WHILE THIS^.fbStations.HasNextObject() DO
	IF __QUERYINTERFACE(THIS^.fbStations.GetNextObject(),ipEachStation) THEN
		//Return TRUE if found
		IF (ipEachStation.TargetGroupe = sStation) OR (ipEachStation.LUID = sStation) THEN
			CheckTargetExists := TRUE;
			EXIT;
		END_IF
	END_IF
END_WHILE

THIS^.fbStations.RestoreIterator();
END_METHOD

METHOD Station : I_XP_Station_PLC
VAR_INPUT
	sLUID : STRING;
END_VAR
//IF no station was found, INTERFACE is 0 -> can generate fatal error
__QUERYINTERFACE(THIS^.fbStations.FindLUID(sLUID),Station);
END_METHOD

METHOD LinkEnvironment : HRESULT
VAR_INPUT
	ipEnvironment : I_CH_Object;
END_VAR

VAR
	ipXpEnvironment : I_XP_Environment;
END_VAR
IF ipEnvironment <> 0 AND_THEN __QUERYINTERFACE(ipEnvironment,ipXpEnvironment) THEN
	THIS^.ipEnvironment := ipXpEnvironment;
ELSE
	LinkEnvironment := E_FAIL;
	THIS^.bErrorDuringFbInit := TRUE;
END_IF
END_METHOD

METHOD LinkGroup : HRESULT
VAR_INPUT
	ipGroup : I_CH_Object;
END_VAR

VAR
	ipXpGroup : I_XP_Group;
END_VAR
IF ipGroup <> 0 AND_THEN __QUERYINTERFACE(ipGroup,ipXpGroup) THEN
	THIS^.ipGroup := ipXpGroup;
ELSE
	LinkGroup := E_FAIL;
	THIS^.bErrorDuringFbInit := TRUE;
END_IF
END_METHOD

METHOD RegisterMover : HRESULT
VAR_INPUT
	ipMover : I_CH_Object;
END_VAR

VAR
	ipXpMover : I_XP_Mover;
END_VAR
IF ipMover = 0 THEN
	//Invalide interface	
	THIS^.bErrorDuringFbInit := TRUE;
	RegisterMover := E_FAIL;
	
ELSIF NOT __QUERYINTERFACE(ipMover, ipXpMover) THEN
	//The required interface is missing
	THIS^.bErrorDuringFbInit := TRUE;
	RegisterMover := E_FAIL;
	
ELSIF THIS^.fbMovers.IsFull THEN
	//List is full
	THIS^.bErrorDuringFbInit := TRUE;
	RegisterMover := E_FAIL;
	
ELSIF THIS^.bInitDone THEN
	//To late. System is initilized
	THIS^.bErrorDuringFbInit := TRUE;
	RegisterMover := E_FAIL;
	
ELSE
	
	THIS^.fbMovers.AddObject(ipMover);
END_IF
END_METHOD

METHOD RegisterStation : HRESULT
VAR_INPUT
	ipStation : I_CH_Object;
END_VAR

VAR
	ipXpStation : I_XP_Station;
END_VAR
IF ipStation = 0 THEN
	//Invalide interface	
	THIS^.bErrorDuringFbInit := TRUE;
	RegisterStation := E_FAIL;
	
ELSIF NOT __QUERYINTERFACE(ipStation, ipXpStation) THEN
	//The required interface is missing
	THIS^.bErrorDuringFbInit := TRUE;
	RegisterStation := E_FAIL;
	
ELSIF THIS^.fbStations.IsFull THEN
	//List is full
	THIS^.bErrorDuringFbInit := TRUE;
	RegisterStation := E_FAIL;
	
ELSIF THIS^.bInitDone THEN
	//To late. System is initilized
	THIS^.bErrorDuringFbInit := TRUE;
	RegisterStation := E_FAIL;
		
ELSE
	
	THIS^.fbStations.AddObject(ipStation);
END_IF
END_METHOD

METHOD RegisterTrack : HRESULT
VAR_INPUT
	ipTrack : I_CH_Object;
END_VAR

VAR
	ipXpTrack : I_XP_Track;
END_VAR
IF ipTrack = 0 THEN
	//Invalide interface	
	THIS^.bErrorDuringFbInit := TRUE;
	RegisterTrack := E_FAIL;
	
ELSIF NOT __QUERYINTERFACE(ipTrack, ipXpTrack) THEN
	//The required interface is missing
	THIS^.bErrorDuringFbInit := TRUE;
	RegisterTrack := E_FAIL;
	
ELSIF THIS^.fbTracks.IsFull THEN
	//List is full
	THIS^.bErrorDuringFbInit := TRUE;
	RegisterTrack := E_FAIL;
	
ELSIF THIS^.bInitDone THEN
	//To late. System is initilized
	THIS^.bErrorDuringFbInit := TRUE;
	RegisterTrack := E_FAIL;
		
ELSE
	
	THIS^.fbTracks.AddObject(ipTrack);
END_IF
END_METHOD

METHOD RegisterTrigger : HRESULT
VAR_INPUT
	ipTrigger	: CHALET_BaseComponents.I_CH_Object;
END_VAR
VAR
	ipXpTrigger : I_Xp_Trigger;
END_VAR
IF ipTrigger = 0 THEN
	//Invalide interface	
	THIS^.bErrorDuringFbInit := TRUE;
	RegisterTrigger := E_FAIL;
	
ELSIF NOT __QUERYINTERFACE(ipTrigger, ipXpTrigger) THEN
	//The required interface is missing
	THIS^.bErrorDuringFbInit := TRUE;
	RegisterTrigger := E_FAIL;
	
ELSIF THIS^.fbTriggers.IsFull THEN
	//List is full
	THIS^.bErrorDuringFbInit := TRUE;
	RegisterTrigger := E_FAIL;
	
ELSIF THIS^.bInitDone THEN
	//To late. System is initilized
	THIS^.bErrorDuringFbInit := TRUE;
	RegisterTrigger := E_FAIL;
		
ELSE
	
	THIS^.fbTriggers.AddObject(ipTrigger);
END_IF
END_METHOD

METHOD RegisterZone : HRESULT
VAR_INPUT
	ipZone	: CHALET_BaseComponents.I_CH_Object;
END_VAR
VAR
	ipXpsZone : I_XP_Zone;
END_VAR
IF ipZone = 0 THEN
	//Invalide interface	
	THIS^.bErrorDuringFbInit := TRUE;
	RegisterZone := E_FAIL;

ELSIF NOT __QUERYINTERFACE(ipZone, ipXpsZone) THEN
	//The required interface is missing
	THIS^.bErrorDuringFbInit := TRUE;
	RegisterZone := E_FAIL;
	
ELSIF THIS^.fbZones.IsFull THEN
	//List is full
	THIS^.bErrorDuringFbInit := TRUE;
	RegisterZone := E_FAIL;
	
ELSIF THIS^.bInitDone THEN
	//To late. System is initilized
	THIS^.bErrorDuringFbInit := TRUE;
	RegisterZone := E_FAIL;
		
ELSE
	
	THIS^.fbZones.AddObject(ipZone);	
END_IF
END_METHOD

{attribute 'monitoring':='call'}
PROPERTY Enviroment : I_XP_Environment
GET
Enviroment := THIS^.ipEnvironment;
END_GET
END_PROPERTY

METHOD FB_init : BOOL
VAR_INPUT
	bInitRetains : BOOL; // if TRUE, the retain variables are initialized (warm start / cold start)
	bInCopyCode : BOOL;  // if TRUE, the instance afterwards gets moved into the copy code (online change)
	
	METAdsPort : UINT; 
END_VAR
VAR
	fbGetCurTaskIdx  : GETCURTASKINDEX;
END_VAR
THIS^.nMETAdsPort := METAdsPort;
END_METHOD

{attribute 'monitoring':='call'}
PROPERTY Feedback : CHALET_BaseComponents.I_CH_Feedback
GET
Feedback := THIS^.fbFeedback;
END_GET
END_PROPERTY

{attribute 'monitoring':='call'}
PROPERTY METAdsPort : UINT
GET
METAdsPort := nMETAdsPort;
END_GET
END_PROPERTY

{attribute 'monitoring':='call'}
PROPERTY Movers : CHALET_BaseComponents.I_CH_LIST
GET
Movers := THIS^.fbMovers;
END_GET
END_PROPERTY

{attribute 'monitoring':='call'}
PROPERTY Stations : CHALET_BaseComponents.I_CH_LIST
GET
Stations := THIS^.fbStations;
END_GET
END_PROPERTY

{attribute 'monitoring':='call'}
PROPERTY Tracks : CHALET_BaseComponents.I_CH_LIST
GET
Tracks := THIS^.fbTracks;
END_GET
END_PROPERTY

{attribute 'monitoring':='call'}
PROPERTY Triggers : CHALET_BaseComponents.I_CH_LIST
GET
Triggers := THIS^.fbTriggers;
END_GET
END_PROPERTY

METHOD Update : HRESULT
VAR_INPUT
END_VAR
VAR
	hr : HRESULT;
END_VAR
//Force to do an init at beginn
IF NOT THIS^.Initialized THEN
	THIS^.Initialize();
	RETURN;
END_IF

hr := S_OK;

hr := GetMostSignificant(hr, THIS^.Enabling());
hr := GetMostSignificant(hr, THIS^.Disabling());




// ********************** Set feedback depending on active command *******************************
IF THIS^.eActiveCommand <> E_NcAxisCommands.None THEN
	fbFeedback.ActiveCommand 	:= TO_STRING(THIS^.eActiveCommand);	
END_IF

CASE THIS^.eActiveCommand OF
	E_NcAxisCommands.None: 
		;

	E_NcAxisCommands.Initialize:
		fbFeedback.Busy 		:= NOT THIS^.bInitDone;
		fbFeedback.Done 		:= THIS^.bInitDone;
		fbFeedback.ErrorId 		:= 0;
		
	E_NcAxisCommands.Enable:
		fbFeedback.Busy 		:= nSeqEnabling > 0;
		fbFeedback.Done 		:= THIS^.Enabled;
		IF nSeqEnabling > 1000 THEN
			fbFeedback.ErrorId 		:= nSeqEnabling;
		END_IF
		
	E_NcAxisCommands.Disable:
		fbFeedback.Busy 		:= nSeqDisabling > 0;
		fbFeedback.Done 		:= THIS^.Disabled;
		IF nSeqDisabling > 1000 THEN
			fbFeedback.ErrorId 		:= nSeqDisabling;
		END_IF
		


	ELSE//External command in subclass
		;
END_CASE


// **********************  Stop to execute commands on .done or .error ***************************
IF fbFeedback.Done OR THIS^.fbFeedback.Error THEN
	eActiveCommand 				:= E_NcAxisCommands.None;
END_IF







hr := GetMostSignificant(hr, THIS^.fbMovers.Update());
hr := GetMostSignificant(hr, THIS^.fbTracks.Update());
hr := GetMostSignificant(hr, THIS^.fbStations.Update());
hr := GetMostSignificant(hr, THIS^.fbZones.Update());
hr := GetMostSignificant(hr, THIS^.fbTriggers.Update());
hr := GetMostSignificant(hr, THIS^.ipGroup.Update());
hr := GetMostSignificant(hr, THIS^.ipEnvironment.Update());


Update:= hr;
END_METHOD

{attribute 'monitoring':='call'}
PROPERTY Zones : CHALET_BaseComponents.I_CH_LIST
GET
Zones := THIS^.fbZones;
END_GET
END_PROPERTY

END_FUNCTION_BLOCK

// COMPONENTs/Track/FB_XP_Track
{attribute 'no_explicit_call' := 'Do not call the body - Stick to OOP'}
(* XPlanar track - n per associated XPlanar. Can be instantiated as an array and/or individually
	The Planar track is a software object that represents a (virtual) one-dimensional path on the two-dimensional XPlanar stator surface. 
	Several Planar movers can be lined up and moved on this path. Collisions are prevented by keeping a preset distance between the movers. *)	
FUNCTION_BLOCK FB_XP_Track EXTENDS FB_CH_Object IMPLEMENTS I_XP_Track
VAR
	//Link to Planar-Track object
	fbTrack : MC_PlanarTrack;
	
	{attribute 'hide'}  
	bInitDone :BOOL := FALSE;
	{attribute 'hide'}               	
	fbFeedback 			: FB_XP_Feedback;
	{attribute 'hide'}                   	
	eActiveCommand 		: CHALET_Nc.E_NcAxisCommands := CHALET_Nc.E_NcAxisCommands.None;
	{attribute 'hide'}
	ipXpSystem : I_XP_System_Registration;
	{attribute 'hide'}	
	nSeqConfiguring : UINT;
	{attribute 'hide'} 
	ipTracksEndAtThis : ARRAY[0..(XPlanarParameterlist.N_MAX_STATIONS_AHEAD_OR_BEHIND-1)] OF I_XP_Track;
	{attribute 'hide'} 
	ipTracksStartFromThis : ARRAY[0..(XPlanarParameterlist.N_MAX_STATIONS_AHEAD_OR_BEHIND-1)] OF I_XP_Track;
	{attribute 'hide'}  
	fbListOfStationsOnTrack : FB_CH_List;
	{attribute 'hide'}  
	bIsClosedLoop : BOOL;
	
	
	{attribute 'hide'}
	fbListOfMoversOnTrack : FB_CH_List;
	{attribute 'hide'}  
	fbTracksAhead : FB_CH_List;
	{attribute 'hide'}  
	fbTracksBehinde : FB_CH_List;
END_VAR

// Planar-Feedback objects
VAR
	{attribute 'hide'} 
	fbFeedbackDisable: MC_PlanarFeedback;
	{attribute 'hide'} 
	fbFeedbackEnable : MC_PlanarFeedback;
	{attribute 'hide'} 
	fbFeedbackAddToGrp : MC_PlanarFeedback;
	{attribute 'hide'} 
	fbFeedbackRmvFromGrp : MC_PlanarFeedback;
	{attribute 'hide'} 
	fbFeedbackReset : MC_PlanarFeedback;
END_VAR

METHOD Configure : HRESULT // This is called once during system enabling
VAR_INPUT
END_VAR
// Validate settings
IF THIS^.Length = 0 THEN
	Configure := E_FAIL;
	THIS^.fbFeedback.LastCommandAccepted:= FALSE;	
	RETURN;
END_IF

THIS^.eActiveCommand 				:= CHALET_NC.E_NcAxisCommands.Configure;
THIS^.fbFeedback.LastCommandAccepted:= TRUE;		
THIS^.fbFeedback.Busy 				:= TRUE;

THIS^.nSeqConfiguring := 10;
Configure := S_OK;
END_METHOD

METHOD Configuring : HRESULT // This is called until S_OK during system enabling
VAR
	ipEachTrackObj : I_CH_Object;
	nIdx : UDINT;
END_VAR
VAR_INST
	fbAdsRead 	: ADSREAD;
	TrackOTCID 	: ARRAY[0..(XPlanarParameterlist.N_MAX_STATIONS_AHEAD_OR_BEHIND-1)] OF OTCID;
END_VAR
VAR CONSTANT
	N_IDX_OFFSET_PREVIOUS_TRACK 	: UDINT := 16#050300D5; // Parameter(online) in Planar Track object
	N_IDX_OFFSET_SUBSEQUENT_TRACK 	: UDINT := 16#050300D6; // Parameter(online) in Planar Track object	
	N_IDX_OFFSET_IS_CLOSED_LOOP		: UDINT := 16#050300E1; // Parameter(online) in Planar Track object	
	
END_VAR
Configuring := S_PENDING;
CASE nSeqConfiguring OF
	0: // Idle
		Configuring := S_OK;
		
	10: //Start
		nSeqConfiguring := 400;
		
		
		
		
		
	//CLOSED LOOP
	400: // Closed loop - Read from Track object
		fbAdsRead.PORT		:= THIS^.ipXpSystem.METAdsPort ; 
		fbAdsRead.IDXGRP	:= THIS^.OID;
		fbAdsRead.IDXOFFS	:= N_IDX_OFFSET_IS_CLOSED_LOOP; 
		fbAdsRead.LEN		:= SIZEOF(THIS^.bIsClosedLoop);
		fbAdsRead.DESTADDR	:= ADR(THIS^.bIsClosedLoop);
			
		fbAdsRead.READ := TRUE;
		nSeqConfiguring := 402;
	
	402: // Wait for reading - Read from Track object
		IF fbAdsRead.ERR THEN
			//Error
			nSeqConfiguring := nSeqConfiguring + 1000;
		ELSIF NOT fbAdsRead.BUSY THEN
			//Done
			nSeqConfiguring := 800;
		END_IF		
		
	

		
	//PREVIOUS_TRACK
	800: // Prepare - Read from Track object
		fbAdsRead.READ := FALSE;
		MEMSET(destAddr := ADR(TrackOTCID), n := SIZEOF(TrackOTCID), fillByte:= 0);
		nSeqConfiguring := 801;
	
	801: // Start read - Read from Track object
		fbAdsRead.PORT		:= THIS^.ipXpSystem.METAdsPort ; 
		fbAdsRead.IDXGRP	:= THIS^.OID;
		fbAdsRead.IDXOFFS	:= N_IDX_OFFSET_PREVIOUS_TRACK; 
		fbAdsRead.LEN		:= SIZEOF(TrackOTCID);
		fbAdsRead.DESTADDR	:= ADR(TrackOTCID);
			
		fbAdsRead.READ := TRUE;
		nSeqConfiguring := 802;
	
	802: // Wait for reading - Read from Track object
		IF fbAdsRead.ERR AND fbAdsRead.ERRID = 6 THEN
			//Error, the reason for this could be that this track has no connected tracks
			//Continous with SUBSEQUENT_TRACK
			nSeqConfiguring := 850;

		ELSIF fbAdsRead.ERR THEN
			//Error
			nSeqConfiguring := nSeqConfiguring + 1000;
		ELSIF NOT fbAdsRead.BUSY THEN
			//Done
			nSeqConfiguring := 803;
		END_IF
	
	803: // Convert to I_XP_Track - Read from Track object
		fbTracksBehinde.Clear();
		FOR nIdx := 0 TO (XPlanarParameterlist.N_MAX_STATIONS_AHEAD_OR_BEHIND-1) DO
			//Get Obj
			ipEachTrackObj := THIS^.ipXpSystem.Tracks.FindOID(TrackOTCID[nIdx]);
			//convert obj -> I_XP_Track
			ToXpTrack(ipEachTrackObj, ipTracksEndAtThis[nIdx]);	
			fbTracksBehinde.AddObject(ipEachTrackObj);
		END_FOR
		nSeqConfiguring := 850;		
	
		
		
		
	//SUBSEQUENT_TRACK	
	850: // Prepare - Read from Track object
		fbAdsRead.READ := FALSE;
		MEMSET(destAddr := ADR(TrackOTCID), n := SIZEOF(TrackOTCID), fillByte:= 0);
		nSeqConfiguring := 851;
	
	851: // Start read - Read from Track object
		fbAdsRead.PORT		:= THIS^.ipXpSystem.METAdsPort ;
		fbAdsRead.IDXGRP	:= THIS^.OID;
		fbAdsRead.IDXOFFS	:= N_IDX_OFFSET_SUBSEQUENT_TRACK;
		fbAdsRead.LEN		:= SIZEOF(TrackOTCID);
		fbAdsRead.DESTADDR	:= ADR(TrackOTCID);
			
		fbAdsRead.READ := TRUE;
		nSeqConfiguring := 852;
	
	852: // Wait for reading - Read from Track object
		IF fbAdsRead.ERR AND fbAdsRead.ERRID = 6 THEN
			//Error, the reason for this could be that this track has no connected tracks
			nSeqConfiguring := 900;
		ELSIF fbAdsRead.ERR THEN
			//Error
			nSeqConfiguring := nSeqConfiguring + 1000;
		ELSIF NOT fbAdsRead.BUSY THEN
			//Done
			nSeqConfiguring := 853;
		END_IF
	
	853: // Convert to I_XP_Track - Read from Track object
		fbTracksAhead.Clear();
		FOR nIdx := 0 TO (XPlanarParameterlist.N_MAX_STATIONS_AHEAD_OR_BEHIND-1) DO
			//Get Obj
			ipEachTrackObj := THIS^.ipXpSystem.Tracks.FindOID(TrackOTCID[nIdx]);
			//convert obj -> I_XP_Track
			ToXpTrack(ipEachTrackObj, ipTracksStartFromThis[nIdx]);	
			fbTracksAhead.AddObject(ipEachTrackObj);
		END_FOR
		nSeqConfiguring := 900;
	
	900: // Config the internal FB_Zone
		nSeqConfiguring := 999;
		
	999: // Done
		Configuring := S_OK;
		
	1000..1999://Error
		Configuring := E_FAIL;
END_CASE


fbAdsRead();
END_METHOD

METHOD Disable : HRESULT
VAR_INPUT
END_VAR
IF NOT THIS^.fbFeedback.Busy THEN
	THIS^.eActiveCommand 				:= CHALET_NC.E_NcAxisCommands.Disable;
	THIS^.fbFeedback.LastCommandAccepted:= TRUE;		
	THIS^.fbFeedback.Busy 				:= TRUE;

	THIS^.fbTrack.Enable(fbFeedbackDisable);
	Disable := S_OK;
ELSE
	Disable := S_FALSE;
	THIS^.fbFeedback.LastCommandAccepted:= FALSE;	
END_IF
END_METHOD

METHOD Enable : HRESULT
VAR_INPUT
END_VAR
IF NOT THIS^.fbFeedback.Busy THEN
	THIS^.eActiveCommand 				:= CHALET_NC.E_NcAxisCommands.Enable;
	THIS^.fbFeedback.LastCommandAccepted:= TRUE;		
	THIS^.fbFeedback.Busy 				:= TRUE;

	THIS^.fbTrack.Enable(fbFeedbackEnable);
	Enable := S_OK;
ELSE
	Enable := S_FALSE;
	THIS^.fbFeedback.LastCommandAccepted:= FALSE;	
END_IF
END_METHOD

METHOD AddToGroup : HRESULT
VAR_INPUT
	iGroup : I_XP_Group;
END_VAR
IF NOT THIS^.fbFeedback.Busy THEN
	THIS^.eActiveCommand 				:= CHALET_NC.E_NcAxisCommands.AddToGroupe;
	THIS^.fbFeedback.LastCommandAccepted:= TRUE;		
	THIS^.fbFeedback.Busy 				:= TRUE;
	
	iGroup.AddTrack(THIS^.fbTrack, THIS^.fbFeedbackAddToGrp);
	AddToGroup := S_OK;
ELSE
	AddToGroup := S_FALSE;
	THIS^.fbFeedback.LastCommandAccepted:= FALSE;	
END_IF
END_METHOD

METHOD RemoveFromGroup : HRESULT
IF NOT THIS^.fbFeedback.Busy THEN
	THIS^.eActiveCommand 				:= CHALET_NC.E_NcAxisCommands.RemoveFromGroupe;
	THIS^.fbFeedback.LastCommandAccepted:= TRUE;		
	THIS^.fbFeedback.Busy 				:= TRUE;
	
	THIS^.fbTrack.RemoveFromGroup(THIS^.fbFeedbackRmvFromGrp);
	
	RemoveFromGroup := S_OK;
ELSE
	RemoveFromGroup := S_FALSE;
	THIS^.fbFeedback.LastCommandAccepted:= FALSE;	
END_IF
END_METHOD

METHOD AddMover : HRESULT
VAR_INPUT
	ipMover : I_XP_Mover;
END_VAR
IF ipMover <> 0 THEN
	AddMover := ipMover.JoinTrack(THIS^);
ELSE
	AddMover := E_FAIL;
END_IF
END_METHOD

{attribute 'monitoring':='call'}
PROPERTY ClosedLoop : BOOL
GET
ClosedLoop := bIsClosedLoop;
END_GET
END_PROPERTY

{attribute 'monitoring':='call'}
PROPERTY CtsMoversOnTrack : UINT
GET
THIS^.Prepare();//Prepare a list movers on this track


CtsMoversOnTrack := TO_UINT(THIS^.fbListOfMoversOnTrack.Size);
END_GET
END_PROPERTY

METHOD FB_init : BOOL
VAR_INPUT
	bInitRetains : BOOL; // if TRUE, the retain variables are initialized (warm start / cold start)
	bInCopyCode : BOOL;  // if TRUE, the instance afterwards gets moved into the copy code (online change)
	
	ipSystem : I_CH_Object;
END_VAR
VAR_INST
	{attribute 'hide'}
	bFBInitCalledOnce : BOOL; //Do the following code once during start up and not during onlinechange
END_VAR
//Do the following code once during start up and not during onlinechange
IF NOT bFBInitCalledOnce THEN 
	
	(* Register to the Xplanar System
	   1. Test if the interface exists
	   2. Test if the object implements a "System for Mover" interface 
	*)
	IF ipSystem <> 0 AND_THEN __QUERYINTERFACE(ipSystem,THIS^.ipXpSystem) THEN
		THIS^.ipXpSystem.RegisterTrack(THIS^);
	END_IF
	

END_IF

bFBInitCalledOnce := TRUE;
END_METHOD

{attribute 'monitoring':='call'}
PROPERTY Feedback : I_XP_Feedback
GET
Feedback := THIS^.fbFeedback;
END_GET
END_PROPERTY

METHOD Initialize : HRESULT
VAR
	hr : HRESULT;
	ipStation : I_XP_Station;
	stVarInfo : __SYSTEM.VAR_INFO;
END_VAR
VAR_INST
	//This error cannot be reset. Requires a reset cold
	{attribute 'hide'}	
	fbInitError : FB_TcAlarm;
END_VAR
// Check if link to track is mapped
IF NOT THIS^.Mapped THEN
	IF NOT fbInitError.bRaised THEN 
		//This error cannot be reset. Requires a reset cold
		fbInitError.CreateEx(stEventEntry:=TC_EVENTS.CHALET_XPlanar_Events.VariableLinkMissing, ipSourceInfo := THIS^.fbSourceInfo, bWithConfirmation := FALSE);
		stVarInfo := __VARINFO(fbTrack);
		fbInitError.ipArguments.AddString(stVarInfo.Symbol);
		fbInitError.Raise(0);
	END_IF
	Initialize := E_FAIL;
	RETURN;
END_IF


IF NOT bInitDone THEN
	//Busy
	Initialize := S_PENDING;
	
	
	//Done as sone list is initilized
	bInitDone := TRUE;
	
ELSE	
	//Done
	Initialize := S_OK;	
END_IF



THIS^.fbFeedback.ActiveCommand 		:= TO_STRING(CHALET_NC.E_NcAxisCommands.Initialize);
THIS^.eActiveCommand 				:= CHALET_NC.E_NcAxisCommands.Initialize;
THIS^.fbFeedback.LastCommandAccepted:= TRUE;	
//Set done or keep in busy state	
THIS^.fbFeedback.HR := Initialize;
END_METHOD

{attribute 'monitoring':='call'}
//[mm]
PROPERTY Length : LREAL
GET
Length := THIS^.fbTrack.GetLength();
END_GET
END_PROPERTY

{attribute 'monitoring':='call'}
PROPERTY Mapped : BOOL //Project is mapped to MC (McToPlc and PlcToMc)
GET
VAR
	bMcToPlcNotMapped 	: BOOL;
END_VAR
bMcToPlcNotMapped := F_GetMappingStatus(ADR(THIS^.fbTrack.MCTOPLC_STD), SIZEOF(THIS^.fbTrack.MCTOPLC_STD)) <> EPlcMappingStatus.MS_Mapped;

Mapped := NOT bMcToPlcNotMapped;
END_GET
END_PROPERTY

{attribute 'monitoring':='call'}
//Unique object ID
PROPERTY OID : OTCID
GET
OID := THIS^.fbTrack.MCTOPLC_STD.TrackOID;
END_GET
END_PROPERTY

{attribute 'monitoring':='call'}
PROPERTY PlanarTrack : REFERENCE TO MC_PlanarTrack
GET
PlanarTrack ref= THIS^.fbTrack;
END_GET
END_PROPERTY

(* Time-critical information is processed here, which can then be polled via the property every cycle. 
The update method is usually at the end of the program and then it is already 'outdated'. *)
METHOD PRIVATE Prepare : HRESULT
VAR
	ipThisTrack : I_XP_Track;
	ipStation : I_XP_Station;
	ipMover : I_XP_Mover;

END_VAR

VAR_INST
	{attribute 'hide'}
	nLastUpdatedCycleCount : UDINT;
END_VAR
//Check if this Cycle the dates are allready prepared
IF nLastUpdatedCycleCount <> TwinCAT_SystemInfoVarList._TaskInfo[THIS^.nTaskIndex].CycleCount THEN
	nLastUpdatedCycleCount := TwinCAT_SystemInfoVarList._TaskInfo[THIS^.nTaskIndex].CycleCount;

	//Creat a list of all Stations on this Track
	ipThisTrack := THIS^;
	THIS^.fbListOfStationsOnTrack.Clear();
	THIS^.ipXpSystem.Stations.ResetIterator();
	WHILE THIS^.ipXpSystem.Stations.HasNextObject() DO
		IF ToXpStation(THIS^.ipXpSystem.Stations.GetNextObject(), ipStation) AND_THEN ipStation.AccocietedTrack <> 0 AND_THEN ipStation.AccocietedTrack = ipThisTrack THEN
			THIS^.fbListOfStationsOnTrack.AddObject(ipStation);
		END_IF
	END_WHILE
	THIS^.ipXpSystem.Stations.RestoreIterator();
	
	
	//Creat a list of all Movers on this Track
	ipThisTrack := THIS^;
	THIS^.fbListOfMoversOnTrack.Clear();
	THIS^.ipXpSystem.Movers.ResetIterator();
	WHILE THIS^.ipXpSystem.Movers.HasNextObject() DO
		IF ToXpMover(THIS^.ipXpSystem.Movers.GetNextObject(), ipMover) AND_THEN ipMover.CurrentTrack <> 0 AND_THEN ipMover.CurrentTrack = ipThisTrack THEN
			THIS^.fbListOfMoversOnTrack.AddObject(ipStation);
		END_IF
	END_WHILE
	THIS^.ipXpSystem.Movers.RestoreIterator();
	
END_IF
END_METHOD

METHOD Reset : HRESULT
VAR_INPUT
END_VAR
THIS^.eActiveCommand 				:= CHALET_NC.E_NcAxisCommands.Reset;
THIS^.fbFeedback.LastCommandAccepted:= TRUE;		
THIS^.fbFeedback.Busy 				:= TRUE;

THIS^.fbTrack.Reset(THIS^.fbFeedbackReset);
Reset := S_OK;
END_METHOD

{attribute 'monitoring':='call'}
//List of interfaces to stations on this track
PROPERTY StationsOnTrack : I_CH_List
GET
VAR
	ipStation : I_XP_Station;
	ipThisTrack : I_XP_Track;
END_VAR
THIS^.Prepare();//Prepare a list stations on this track

StationsOnTrack := THIS^.fbListOfStationsOnTrack;
END_GET
END_PROPERTY

{attribute 'monitoring':='call'}
//List of interfaces from other tracks
PROPERTY TracksAhead : I_CH_List
GET
TracksAhead := fbTracksAhead;
END_GET
END_PROPERTY

{attribute 'monitoring':='call'}
//List of interfaces from other tracks
PROPERTY TracksBehinde : I_CH_List
GET
TracksBehinde:= fbTracksBehinde;
END_GET
END_PROPERTY

{attribute 'monitoring':='call'}
//zzz Todo Delet me
PROPERTY TracksEndAtThis : REFERENCE TO  ARRAY[0..(XPlanarParameterlist.N_MAX_STATIONS_AHEAD_OR_BEHIND-1)] OF I_XP_Track
GET
TracksEndAtThis REF= ipTracksEndAtThis;
END_GET
END_PROPERTY

{attribute 'monitoring':='call'}
PROPERTY TracksStartFromThis : REFERENCE TO ARRAY[0..(XPlanarParameterlist.N_MAX_STATIONS_AHEAD_OR_BEHIND-1)] OF I_XP_Track
GET
TracksStartFromThis REF= ipTracksStartFromThis;
END_GET
END_PROPERTY

METHOD PUBLIC Update : HRESULT
VAR_INPUT
END_VAR



// ********************** Set feedback depending on active command *******************************
IF THIS^.eActiveCommand <> E_NcAxisCommands.None THEN
	fbFeedback.ActiveCommand 	:= TO_STRING(THIS^.eActiveCommand);	
END_IF

CASE THIS^.eActiveCommand OF
	E_NcAxisCommands.None: 
		//Display if a Mover Error is active during no command is active
		IF THIS^.fbTrack.Error AND NOT fbFeedback.Error THEN 
			fbFeedback.ErrorId 			:= THIS^.fbTrack.ErrorID;
			fbFeedback.ActiveCommand 	:= TO_STRING(E_NcAxisCommands.None);	
			fbFeedback.ClearObjectInfo();
		END_IF

	E_NcAxisCommands.Initialize:
		fbFeedback.Busy 			:= NOT THIS^.bInitDone;
		fbFeedback.Done 			:= THIS^.bInitDone;
		fbFeedback.ErrorId 			:= 0;
		fbFeedback.ClearObjectInfo();
		                        	
	E_NcAxisCommands.Enable:     	
		fbFeedback.Busy 			:= fbFeedbackEnable.Busy;
		fbFeedback.Done 			:= fbFeedbackEnable.Done;
		fbFeedback.ErrorId 			:= fbFeedbackEnable.ErrorID;
        fbFeedback.ObjectInfo		:= fbFeedbackEnable.objectInfo;
                                			                        	
	E_NcAxisCommands.Disable:     	
		fbFeedback.Busy 			:= fbFeedbackDisable.Busy;
		fbFeedback.Done 			:= fbFeedbackDisable.Done;
		fbFeedback.ErrorId 			:= fbFeedbackDisable.ErrorID;
        fbFeedback.ObjectInfo		:= fbFeedbackDisable.objectInfo;
		
	E_NcAxisCommands.Configure:
		fbFeedback.Busy 		:= nSeqConfiguring > 0;
		fbFeedback.Done 		:= nSeqConfiguring = 999;
		IF nSeqConfiguring > 1000 THEN
			fbFeedback.ErrorId 		:= nSeqConfiguring;
		END_IF
                                			                        	
	E_NcAxisCommands.Reset:     	
		fbFeedback.Busy 			:= fbFeedbackReset.Busy;
		fbFeedback.Done 			:= fbFeedbackReset.Done;
		fbFeedback.ErrorId 			:= fbFeedbackReset.ErrorID;
        fbFeedback.ObjectInfo		:= fbFeedbackReset.objectInfo;
                                      			                        	
	E_NcAxisCommands.AddToGroupe:     	
		fbFeedback.Busy 			:= fbFeedbackAddToGrp.Busy;
		fbFeedback.Done 			:= fbFeedbackAddToGrp.Done;
		fbFeedback.ErrorId 			:= fbFeedbackAddToGrp.ErrorID;
        fbFeedback.ObjectInfo		:= fbFeedbackAddToGrp.objectInfo;
                                      			                        	
	E_NcAxisCommands.RemoveFromGroupe:     	
		fbFeedback.Busy 			:= fbFeedbackRmvFromGrp.Busy;
		fbFeedback.Done 			:= fbFeedbackRmvFromGrp.Done;
		fbFeedback.ErrorId 			:= fbFeedbackRmvFromGrp.ErrorID;
        fbFeedback.ObjectInfo		:= fbFeedbackRmvFromGrp.objectInfo;
                                		
	ELSE//External command in subclass
		;
END_CASE


// **********************  Stop to execute commands on .done or .error ***************************
IF fbFeedback.Done OR THIS^.fbFeedback.Error THEN
	eActiveCommand 				:= E_NcAxisCommands.None;
END_IF

//Update xplanar object
THIS^.fbTrack.Update();

//Update feedback object
fbFeedbackEnable.Update(); 
fbFeedbackDisable.Update(); 
fbFeedbackReset.Update(); 
fbFeedbackAddToGrp.Update(); 
fbFeedbackRmvFromGrp.Update();
END_METHOD

END_FUNCTION_BLOCK

// COMPONENTs/Track/I_XP_Track_PLC
INTERFACE I_XP_Track_PLC EXTENDS __SYSTEM.IQueryInterface

{attribute 'monitoring':='call'}
PROPERTY CtsMoversOnTrack : UINT
GET
END_GET
END_PROPERTY

{attribute 'monitoring':='call'}
PROPERTY Feedback : I_XP_Feedback
GET
END_GET
END_PROPERTY

{attribute 'monitoring':='call'}
//[mm]
PROPERTY Length : LREAL
GET
END_GET
END_PROPERTY

{attribute 'monitoring':='call'}
PROPERTY Mapped : BOOL //Project is mapped to MC (McToPlc and PlcToMc)
GET
END_GET
END_PROPERTY

{attribute 'monitoring':='call'}
//Unique object ID
PROPERTY OID : OTCID
GET
END_GET
END_PROPERTY

{attribute 'monitoring':='call'}
PROPERTY PlanarTrack : REFERENCE TO MC_PlanarTrack
GET
END_GET
END_PROPERTY

{attribute 'monitoring':='call'}
//List of interfaces to stations on this track
PROPERTY StationsOnTrack : I_CH_List
GET
END_GET
END_PROPERTY

{attribute 'monitoring':='call'}
//List of interfaces from other tracks
PROPERTY TracksAhead : I_CH_List
GET
END_GET
END_PROPERTY

{attribute 'monitoring':='call'}
//List of interfaces from other tracks
PROPERTY TracksBehinde : I_CH_List
GET
END_GET
END_PROPERTY

{attribute 'monitoring':='call'}
PROPERTY TracksEndAtThis : REFERENCE TO  ARRAY[0..(XPlanarParameterlist.N_MAX_STATIONS_AHEAD_OR_BEHIND-1)] OF I_XP_Track
GET
END_GET
END_PROPERTY

{attribute 'monitoring':='call'}
PROPERTY TracksStartFromThis : REFERENCE TO ARRAY[0..(XPlanarParameterlist.N_MAX_STATIONS_AHEAD_OR_BEHIND-1)] OF I_XP_Track
GET
END_GET
END_PROPERTY

END_INTERFACE
